FUNCTION_BLOCK FB_PythonScript
VAR_INPUT
	i_sScriptName		:STRING;
	i_sScriptPath		:STRING;
	i_sScriptDir		:STRING;
	i_bStart			:BOOL;
END_VAR
VAR_IN_OUT
	iq_bScriptBusy		:BOOL;
	iq_bScriptDone		:BOOL;
	iq_bScriptError		:BOOL;
	iq_sScriptError		:STRING;
END_VAR
VAR_OUTPUT
	q_bBusy				:BOOL;
	q_bError			:BOOL;
	q_bDone				:BOOL;
	q_sStatus			:STRING;
END_VAR
VAR
	ntProcess			:NT_StartProcess;
	bStartNT			:BOOL;

	iStep				:INT;
	tTimeOut_TON1		:TON;
	tTimeOut1			:TIME;
	tTimeOut_TON2		:TON;
	tTimeOut2			:TIME;
END_VAR

ACT_StartProcess();

tTimeOut1:=T#30S;
tTimeOut2:=T#30S;

q_sStatus:=iq_sScriptError;

CASE iStep OF
	
	0:

		q_bBusy:=FALSE;
		tTimeOut_TON1(IN:=FALSE,PT:=tTimeOut1);
		tTimeOut_TON2(IN:=FALSE,PT:=tTimeOut2);
	
		IF i_bStart THEN
			q_bError:=FALSE;
			q_bDone:=FALSE;
			q_bBusy:=TRUE;
			
			iq_bScriptBusy:=FALSE;
			iq_bScriptDone:=FALSE;
			iq_bScriptError:=FALSE;
			iq_sScriptError:='';
			
			iStep:=10;
		END_IF
	
	10:
		bStartNT:=TRUE;
		IF ntProcess.BUSY THEN
			iStep:=15;
		END_IF
	
	15:
		IF NOT ntProcess.BUSY THEN
			iStep:=20;
		ELSIF ntProcess.ERR THEN
			iStep:=999;
		END_IF
	20:
		tTimeOut_TON1(IN:=TRUE,PT:=tTimeOut1);
		IF NOT iq_bScriptDone AND NOT iq_bScriptError THEN
			iStep:=30;
		ELSIF tTimeOut_TON1.Q OR iq_bScriptError THEN
			iStep:=999;
		END_IF
	30:
		tTimeOut_TON2(IN:=TRUE,PT:=tTimeOut2);
		IF iq_bScriptDone AND NOT iq_bScriptError THEN 
			iStep:=50;	
		ELSIF tTimeOut_TON2.Q OR iq_bScriptError THEN
			iStep:=999;
		END_IF
		
	50:
		q_bDone:=TRUE;
		iStep:=0;
	999:
		
		q_bError:=TRUE;
		iStep:=0;
		
		
END_CASE

ACTION ACT_StartProcess:
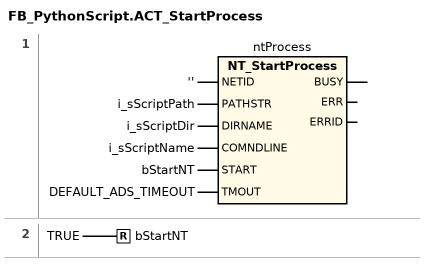
// NETWORK 1
ntProcess(
    NETID := '',
    PATHSTR := i_sScriptPath,
    DIRNAME := i_sScriptDir,
    COMNDLINE := i_sScriptName,
    START := bStartNT,
    TMOUT := DEFAULT_ADS_TIMEOUT); // NT_StartProcess

// NETWORK 2
bStartNT R= TRUE;
END_ACTION

END_FUNCTION_BLOCK

(* stored: Version 1.1.0.1, ProductVersion 3.1.4024.12
   POU FB_PythonScript: Id {fbc4a31d-6df8-4873-a5db-6f39f4daff21}, SpecialFunc None
   Action ACT_StartProcess: Id {84a73c2c-4e2d-4e6a-91f5-23f0553e2a30} *)
